# B&R Automation Studio project Robot_control
Automation Studio 4.8.2.72

## Configuration Config1

CPU X20CP1382, AutomationRuntime B4.82, Build 4.1.2, Vc V4.72.1

### Task classes (Cpu.sw)
```
Cyclic#1 (cycle 1000 us, tolerance 1000 us):
  Program <- Program.prg
  OpcUA <- OpcUA.prg
  TCPServer <- TCPServer.prg
Binaries: udbdef, FWRules, TCData, sysconf, Role, User, iomap, ashwd, asfw, arconfig, ashwac
Libraries: AsIecCon, AsOpcUac, AsOpcUas, AsTCP, AsBrStr, runtime, astime, standard
```

### Hardware
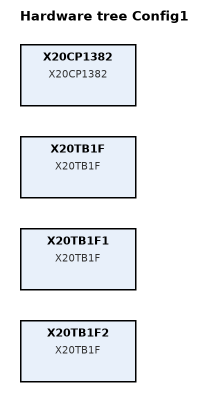
```
X20CP1382 : X20CP1382 v1.10.0.0  [X1 -> X1.SL; X2 -> X2.SL; X3 -> X3.SL]
  Module X1 (Type=X1, Virtual=true, Version=1.10.0.0)
    Connection (Connector=SS1, TargetModule=X20TB1F, TargetConnector=SS)
    Connection (Connector=SL, TargetModule=X20CP1382, TargetConnector=X1)
  Module X2 (Type=X2, Virtual=true, Version=1.10.0.0)
    Connection (Connector=SS1, TargetModule=X20TB1F1, TargetConnector=SS)
    Connection (Connector=SL, TargetModule=X20CP1382, TargetConnector=X2)
  Module X3 (Type=X3, Virtual=true, Version=1.10.0.0)
    Connection (Connector=SS1, TargetModule=X20TB1F2, TargetConnector=SS)
    Connection (Connector=SL, TargetModule=X20CP1382, TargetConnector=X3)
  Connector IF2:
    ActivateDevice = 1
    Mode = Manual
    InternetAddress = 192.168.0.20
    SubnetMask = 255.255.255.0
    ActivateSnmp = 2
  Connector IF7:
    Timeout = 1
  ConfigurationID = robot_control_Config1
  SystemTick = 1000
  TaskClassIdleTime = 1000
  Cyclic1Duration = 1000
  Cyclic1Tolerance = 1000
  Cyclic2Duration = 2000
  Cyclic2Tolerance = 2000
X20TB1F : X20TB1F v1.0.0.0
X20TB1F1 : X20TB1F v1.0.0.0
X20TB1F2 : X20TB1F v1.0.0.0
```

### IoMap.iom - X20CP1382/IoMap.iom
```iecst
VAR_CONFIG
	::Program:this.M1.direction AT %QX."X3".DigitalOutput04;
	::Program:this.M1.freq AT %QX."X3".DigitalOutput09;
	::Program:this.M2.direction AT %QX."X3".DigitalOutput05;
	::Program:this.M3.direction AT %QX."X3".DigitalOutput06;
	::Program:this.M2.freq AT %QX."X3".DigitalOutput10;
	::Program:this.M3.freq AT %QX."X3".DigitalOutput11;
	::Program:this.btn1.pressed AT %IX."X1".DigitalInput03;
	::Program:this.btn2.pressed AT %IX."X1".DigitalInput02;
	::Program:this.btn4.pressed AT %IX."X1".DigitalInput04;
	::Program:this.btn3.pressed AT %IX."X1".DigitalInput01;
	::Program:this.pencilSharp AT %QX."X3".DigitalOutput08;
	gNettime  AT %ID."X20CP1382".IF6.Nettime;
END_VAR
```

## Logical view

Binary libraries used (declarations not repeated): operator, runtime, astime, AsIecCon, AsOpcUac, AsOpcUas, AsTCP, AsBrStr, standard

### Global.typ
```iecst
TYPE
	coord_typ : 	STRUCT  (*Meant to be an array of coordinates*)
		z : DINT; (*Also called draw*)
		y : DINT;
		x : DINT;
	END_STRUCT;
END_TYPE
```

### Global.var
```iecst
VAR
	coord : ARRAY[0..LENGT_OF_COORD] OF coord_typ;
	gNettime : DINT;
	pSharp : BOOL;
	draw_old : DINT;
	draw : DINT := 0;
	y_coord : DINT := 0;
	x_coord : DINT := 0;
	goTo : STRING[80];
END_VAR
(*SPEED : TIME;*)
(*Global constants*)
VAR CONSTANT
	LENGT_OF_COORD : USINT := 200; (*maximum number of stored coords*)
END_VAR
```

### Program Logical/OpcUA

#### Types.typ
```iecst
TYPE
	OPC :
		(
		OPC_START_OPERATE,
		OPC_METHOD_CALLED,
		OPC_METHOD_EXECUTE,
		OPC_FINISH_OPERATE,
		OPC_FINISH_METHOD,
		OPC_ERROR
		);
END_TYPE
```

#### Variables.var
```iecst
VAR
	lookAt : USINT;
	result : USINT;
	ma : USINT;
	mb : USINT;
	UaSrv_MethodOperate_0 : UaSrv_MethodOperate;
	stOpcMethod : OPC;
	errorID : DWORD;
END_VAR
```

#### Main.st
```iecst
PROGRAM _INIT

END_PROGRAM

PROGRAM _CYCLIC
	CASE stOpcMethod OF
		OPC_START_OPERATE: // start operate
			UaSrv_MethodOperate_0.Action  := UaMoa_CheckIsCalled;
			UaSrv_MethodOperate_0.MethodName := 'Multiply';
			UaSrv_MethodOperate_0.Execute := TRUE;
			stOpcMethod := OPC_METHOD_CALLED;
		OPC_METHOD_CALLED: // check if method called
			UaSrv_MethodOperate_0();
			IF UaSrv_MethodOperate_0.Busy THEN
				UaSrv_MethodOperate_0.Execute := FALSE;
			ELSE
				IF UaSrv_MethodOperate_0.Done THEN
					errorID := 0;
					IF UaSrv_MethodOperate_0.IsCalled THEN
						stOpcMethod := OPC_METHOD_EXECUTE; // method is called
					END_IF
					UaSrv_MethodOperate_0.Execute := TRUE;
				END_IF
				IF UaSrv_MethodOperate_0.Error THEN
					errorID:= UaSrv_MethodOperate_0.ErrorID;
					stOpcMethod := OPC_ERROR;
				END_IF
			END_IF
		OPC_METHOD_EXECUTE: // execute method code
			result := ma * mb;
			stOpcMethod := OPC_FINISH_OPERATE;
		OPC_FINISH_OPERATE: // finish operate
			UaSrv_MethodOperate_0.Action  := UaMoa_Finished;
			UaSrv_MethodOperate_0.MethodName := 'Multiply';
			UaSrv_MethodOperate_0.Execute := TRUE;
			stOpcMethod := OPC_FINISH_METHOD;
		OPC_FINISH_METHOD: // finish method
			UaSrv_MethodOperate_0();
			IF UaSrv_MethodOperate_0.Busy THEN
				UaSrv_MethodOperate_0.Execute := FALSE;
			ELSE
				IF UaSrv_MethodOperate_0.Done THEN
					errorID:= 0;
					stOpcMethod := OPC_START_OPERATE; // method is finished, wait again for call
				END_IF
				IF UaSrv_MethodOperate_0.Error THEN
					errorID:= UaSrv_MethodOperate_0.ErrorID;
					stOpcMethod := OPC_ERROR;
				END_IF
			END_IF
	END_CASE;
END_PROGRAM

PROGRAM _EXIT

END_PROGRAM
```

- Methods.uam (not shown)

### Program Logical/Program (IEC)

#### Main.st - Init, cyclic, exit code
```iecst
PROGRAM _INIT
	draw := 5;
	this.start := TRUE;
	this.topSpeed 		:= T#0ms; 	// This parameter will slow the topspeed of all axis.
	this.acceleration	:= 1;		// This parameter will smoothen the acceleration of all axis.

END_PROGRAM

PROGRAM _CYCLIC
	(**********************************************************************************************)
	(************************************** Startup sequence **************************************)
	(**********************************************************************************************)
	IF this.start AND gNettime <> 0 THEN
		CASE this.startCase OF
			0: // First find M3 and M2 home switch
				this.M3.backward 	:= TRUE;
				this.M2.backward 	:= TRUE;

				IF this.btn3.pressed THEN
					this.M1.backward:= TRUE;
					this.startCase 	:= 10;
				END_IF;

			10: // Waiting for M1 and M2 to be homed
				IF this.btn1.pressed THEN
					this.M1.counter	:= 0;
				END_IF;

				IF this.btn2.pressed THEN
					this.M2.counter := 0;
				END_IF;

				IF this.btn1.pressed AND this.btn2.pressed THEN
					this.startCase := 15;
				END_IF;

			15:// going to origo (0,0)
				IF this.M1.counter < 4000 THEN
					this.M1.forward := TRUE;
				ELSE
					this.M1.forward := FALSE;
				END_IF;

				IF this.M2.counter < 275 THEN
					this.M2.forward := TRUE;
				ELSE
					this.M2.forward := FALSE;
				END_IF;

				IF this.M1.counter >= 4000 AND this.M2.counter >= 275 THEN
					this.startCase := 20;
				END_IF;

			20: // make sure the pencil have reached origo with M3
				IF this.btn4.pressed THEN
					this.startCase := 25;
				ELSE
					this.M3.forward := TRUE;
				END_IF;

			25: // Set all counter values to 0
				this.M1.counter := 0;
				this.M2.counter := 0;
				this.M3.counter := 0;
				this.startCase := 30;

			30: // Lift the pencil from the paper again
				IF this.M3.counter > -500 THEN
					this.M3.backward := TRUE;
				ELSE
					this.M3.backward := FALSE;
					this.startCase := 35;
				END_IF;

			35: // Ready to start drawing
				this.start 		:= FALSE;
				this.startCase 	:= FALSE;
				this.isReady 	:= TRUE;

		END_CASE;
	END_IF

	(**********************************************************************************************)
	(*********************************** Coordinate translation ***********************************)
	(**********************************************************************************************)
	// Read and translate the coordinates from java server
	IF NOT pSharp THEN
		CASE case_draw OF
			0: // start the case
				IF coord[LENGT_OF_COORD].x <> -1 AND coord[LENGT_OF_COORD].y <> -1 AND coord[LENGT_OF_COORD].z <> -1 THEN
					this.coord.x := coord[LENGT_OF_COORD].x;
					this.coord.y := coord[LENGT_OF_COORD].y;
					this.coord.z := coord[LENGT_OF_COORD].z;
					coord[LENGT_OF_COORD].x := -1;
					coord[LENGT_OF_COORD].y := -1;
					coord[LENGT_OF_COORD].z := -1;
					case_draw := 5;
				END_IF

			5: // which height should we goto?
				IF this.coord.z = 0 THEN // Black
					this.M3.goToCounter := 110;
					this.M3.goTo 		:= TRUE;
				ELSIF this.coord.z = 1 THEN
					this.M3.goToCounter := 75;
					this.M3.goTo 		:= TRUE;
				ELSIF this.coord.z = 2 THEN
					this.M3.goToCounter := 30;
					this.M3.goTo 		:= TRUE;
				ELSIF this.coord.z = 3 THEN
					this.M3.goToCounter := -65;
					this.M3.goTo 		:= TRUE;
				ELSIF this.coord.z = 4 THEN
					this.M3.goToCounter := -75;
					this.M3.goTo 		:= TRUE;
				ELSIF this.coord.z = 5 THEN // White
					this.M3.goToCounter := -200;
					this.M3.goTo 		:= TRUE;
				END_IF

				IF this.M3.counter = this.M3.goToCounter THEN
					case_draw := 10;
				END_IF

			10: // Goto all the coordinates, and then go back to state 0 to calculate next coordinate
				this.M1.goToCounter := this.coord.x * 40;
				this.M2.goToCounter := this.coord.y * 40;
				this.M1.goTo := TRUE;
				this.M2.goTo := TRUE;
				IF this.M3.counter <> this.M3.goToCounter THEN
					this.M3.goTo := TRUE;
				END_IF

				IF (this.M1.goToCounter = this.M1.counter AND this.M2.goToCounter = this.M2.counter AND this.M3.goToCounter = this.M3.counter) THEN
					case_draw := 0;
				END_IF

		END_CASE;
	END_IF;

	(**********************************************************************************************)
	(*********************************** Pencil sharpener logic ***********************************)
	(**********************************************************************************************)
	// Controls the acceleration when pencil sharpening
	IF EDGEPOS(pSharp) AND this.acceleration < 2 THEN
		this.acceleration 			:= this.acceleration + 2;
		this.accelerationChangePS 	:= TRUE;
	ELSIF EDGENEG(pSharp) AND this.accelerationChangePS THEN
		this.acceleration			:= this.acceleration - 2;
		this.accelerationChangePS	:= FALSE;
	END_IF

	// Calculate when to sharp the pencil
	// No wear on the pencil when draw value is 5
	// Approx. 175000 ms if the pencil draw value is 4
	// Approx. 164000 ms if the pencil draw value is 3
	// Approx. 150000 ms if the pencil draw value is 2
	// Approx. 130000 ms if the pencil draw value is 1
	// Approx. 100000 ms if the pencil draw value is 0
	IF this.coord.x > 0 AND this.coord.y > 0 AND this.coord.z > 0 THEN
		IF draw = 4 THEN
			dull_counter := dull_counter + 1;
		ELSIF draw = 3 THEN
			dull_counter := dull_counter + 1.06;
		ELSIF draw = 2 THEN
			dull_counter := dull_counter + 1.16;
		ELSIF draw = 1 THEN
			dull_counter := dull_counter + 1.35;
		ELSIF draw = 0 THEN
			dull_counter := dull_counter + 1.75;
		END_IF
	END_IF

	IF (dull_counter > 175000) THEN
		pSharp := TRUE;
		dull_counter := 0;
		this.startPS := TRUE;
	END_IF;

	IF this.startPS THEN // When the dull counter runs out, pencil sharpener case starts
		CASE this.startPSCase OF
			0: // Store goTo values
				this.M1.goToCounter := this.M1.counter;
				this.M3.goToCounter := this.M3.counter;
				this.m3TempPS		:= this.M3.counter;
				this.startPSCase := 5;

			5: // lift the pencil from the drawing plane, and go to an height that fits the pencil sharpener
				this.M3.backward := TRUE;

				IF this.M3.counter < -200 AND this.M1.counter > -2500 THEN
					this.M1.backward := TRUE;
				ELSE
					this.M1.backward := FALSE;
				END_IF

				IF this.M3.counter = -3200 THEN
					this.M3.backward := FALSE;
					this.startPSCase := 10;
				END_IF

			10: // Start moving towards the pencil sharpener, and wait for switch above pencil sharpener to be activated
				this.M1.backward := TRUE;
				IF this.btn1.pressed THEN
					this.M1.backward := FALSE;
					this.startPSCase := 15;
				END_IF

			15: // start pencil sharpener, and go into the pencil sharpener
				this.pencilSharp := TRUE;
				this.M3.goToCounter := 110;
				this.M3.goTo := TRUE;

				IF EDGEPOS(this.btn4.pressed)THEN
					this.M3.counter	:= 0;
				END_IF

				IF this.btn4.pressed THEN
					sharp_counter := sharp_counter +1;
				END_IF

				IF sharp_counter > 500 THEN // go deeper
					sharp_counter := 0;
					this.startPSCase := 16;
				END_IF;

			16: // start going deeper
				this.M3.goToCounter := 130;
				this.M3.goTo := TRUE;
				sharp_counter := sharp_counter +1;

				IF sharp_counter > 500 THEN // go deeper
					sharp_counter := 0;
					this.startPSCase := 17;
				END_IF;

			17: // start going deeper
				this.M3.goToCounter := 145;
				this.M3.goTo := TRUE;
				sharp_counter := sharp_counter +1;

				IF sharp_counter > 3000 THEN // retreat
					sharp_counter := 0;
					this.startPSCase := 20;
				END_IF;

			20: // move out of the pencil sharpener
				this.M3.backward := TRUE;

				IF this.M3.counter = -1950 THEN
					this.M3.backward := FALSE;
					this.startPSCase := 25;
					this.pencilSharp := FALSE;
				END_IF

			25: // move back to position
				this.M1.goTo := TRUE;

				IF this.M1.counter > - 2800 THEN
					this.M3.goToCounter := 800;
					this.M3.goTo 		:= TRUE;
					this.startPSCase 	:= 27;
				END_IF

			27: // Calibrate axis 3 on the drawining plane
				IF this.M1.goTo = FALSE AND this.M3.goTo = FALSE THEN
					this.M3.forward := TRUE;
				END_IF

				IF this.btn4.pressed THEN
					this.M3.counter 	:= 0;
					this.M3.forward		:= FALSE;
					this.startPSCase 	:= 30;
				END_IF

			30: // go to the correct heigt
				IF this.M1.goTo = FALSE THEN
					this.M3.goToCounter := this.m3TempPS;
					this.M3.goTo := TRUE;
					this.startPSCase := 35;
				END_IF

			35: // Continues from where it left
				this.startPS := FALSE;
				this.startPSCase := 0;
				pSharp := FALSE;

		END_CASE
	END_IF

	(**********************************************************************************************)
	(****************************************** Subcasses *****************************************)
	(**********************************************************************************************)
	M1_speedCase;
	M2_speedCase;
	M3_speedCase;

END_PROGRAM
```

#### Types.typ - Local data types
```iecst
TYPE
	m_typ : 	STRUCT  (*Types used for all motors*)
		endSwitch : BOOL;
		freq : BOOL; (*Output frequency for the steppermotor*)
		backward : BOOL; (*Backward movement towards the switch when true*)
		forward : BOOL; (*Forward movement when true*)
		direction : BOOL; (*Output direction for the steppermotor*)
		counter : DINT; (*Actual position*)
		goTo : BOOL; (*When true, the axis will goTo the goToCounter value*)
		goToCounter : DINT; (*The postion the axis should go to*)
		speedCaseTON : TON; (*Used to control acceleration*)
		speedCase : USINT; (*Used to control acceleration*)
		overRideCase : USINT; (*This case is used if you want to go further than the endswitch*)
	END_STRUCT;
	this_typ : 	STRUCT  (*Local structure type*)
		M1 : m_typ;
		M2 : m_typ;
		M3 : m_typ;
		topSpeed : TIME; (*T#0ms = 1 bit every 1 ms, T#5ms = 1 bit every 5 ms*)
		acceleration : USINT; (*0 = instant topspeed, 10 = slowest acceleration*)
		btn2 : btn_typ;
		isReady : BOOL;
		btn4 : btn_typ;
		btn3 : btn_typ;
		btn1 : btn_typ;
		startCase : USINT;
		start : BOOL;
		startPSCase : USINT;
		startPS : BOOL;
		accelerationChangePS : BOOL; (*If the acceleration have been changed when pencil sharpening, then this bool will be true*)
		m3TempPS : DINT;
		pencilSharp : BOOL;
		greyScale : USINT;
		print : BOOL; (*If print is equal to 1 then it should be printing*)
		coord : coord_typ;
	END_STRUCT;
	btn_typ : 	STRUCT
		pressed : BOOL;
	END_STRUCT;
END_TYPE
```

#### Variables.var - Local variables
```iecst
VAR
	dull_counter : REAL;
	sharp_counter : DINT;
	case_draw : USINT;
	this : this_typ;
END_VAR
```

#### M1_speedCase.st
```iecst
ACTION M1_speedCase:

	CASE this.M1.speedCase OF
		0: // highest speed
			this.M1.speedCaseTON.PT := this.topSpeed;

		1:
			this.M1.speedCaseTON.PT := this.topSpeed + T#1ms;

		2:
			this.M1.speedCaseTON.PT := this.topSpeed + T#2ms;

		3:
			this.M1.speedCaseTON.PT := this.topSpeed + T#3ms;

		4:
			this.M1.speedCaseTON.PT := this.topSpeed + T#4ms;

		5:
			this.M1.speedCaseTON.PT := this.topSpeed + T#5ms;

		6:
			this.M1.speedCaseTON.PT := this.topSpeed + T#6ms;

		7:
			this.M1.speedCaseTON.PT := this.topSpeed + T#7ms;

		8:
			this.M1.speedCaseTON.PT := this.topSpeed + T#8ms;

		9:
			this.M1.speedCaseTON.PT := this.topSpeed + T#9ms;

		10:
			this.M1.speedCaseTON.PT := this.topSpeed + T#10ms;

	END_CASE

	IF this.M1.forward OR this.M1.backward THEN
		IF this.M1.speedCaseTON.Q THEN
			this.M1.speedCaseTON.IN := FALSE;

			IF this.M1.freq THEN
				this.M1.freq 		:= FALSE;
			ELSE
				this.M1.freq		:= TRUE;
			END_IF

		ELSE
			this.M1.speedCaseTON.IN := TRUE;

		END_IF
	END_IF

	IF this.M1.forward THEN
		this.M1.direction := TRUE;

		IF EDGEPOS(this.M1.freq) THEN
			this.M1.counter := this.M1.counter + 1;

			IF this.M1.speedCase > 0 THEN
				this.M1.speedCase := this.M1.speedCase - 1;
			END_IF

		ELSIF EDGEPOS(NOT(this.M1.freq)) THEN
			this.M1.counter := this.M1.counter + 1;
		END_IF;
	ELSIF this.M1.backward THEN
		this.M1.direction := FALSE;

		IF EDGEPOS(this.M1.freq) THEN
			this.M1.counter := this.M1.counter - 1;

			IF this.M1.speedCase > 0 THEN
				this.M1.speedCase := this.M1.speedCase - 1;
			END_IF

		ELSIF EDGEPOS(NOT(this.M1.freq)) THEN
			this.M1.counter := this.M1.counter - 1;
		END_IF;

	END_IF
	IF EDGEPOS(NOT(this.M1.backward)) OR EDGEPOS(NOT(this.M1.forward)) THEN
		this.M1.speedCase := this.acceleration;

	END_IF

	this.M1.speedCaseTON ();
END_ACTION
```

#### M2_speedCase.st
```iecst
ACTION M2_speedCase:

	CASE this.M2.speedCase OF
		0: // highest speed
			this.M2.speedCaseTON.PT := this.topSpeed;

		1:
			this.M2.speedCaseTON.PT := this.topSpeed + T#1ms;

		2:
			this.M2.speedCaseTON.PT := this.topSpeed + T#2ms;

		3:
			this.M2.speedCaseTON.PT := this.topSpeed + T#3ms;

		4:
			this.M2.speedCaseTON.PT := this.topSpeed + T#4ms;

		5:
			this.M2.speedCaseTON.PT := this.topSpeed + T#5ms;

		6:
			this.M2.speedCaseTON.PT := this.topSpeed + T#6ms;

		7:
			this.M2.speedCaseTON.PT := this.topSpeed + T#7ms;

		8:
			this.M2.speedCaseTON.PT := this.topSpeed + T#8ms;

		9:
			this.M2.speedCaseTON.PT := this.topSpeed + T#9ms;

		10:
			this.M2.speedCaseTON.PT := this.topSpeed + T#10ms;

	END_CASE

	IF this.M2.forward OR this.M2.backward THEN
		IF this.M2.speedCaseTON.Q THEN
			this.M2.speedCaseTON.IN := FALSE;

			IF this.M2.freq THEN
				this.M2.freq 		:= FALSE;
			ELSE
				this.M2.freq		:= TRUE;
			END_IF

		ELSE
			this.M2.speedCaseTON.IN := TRUE;

		END_IF
	END_IF

	IF this.M2.forward THEN // Logic for acceleration
		this.M2.direction := TRUE;

		IF EDGEPOS(this.M2.freq) THEN
			this.M2.counter := this.M2.counter + 1;

			IF this.M2.speedCase > 0 THEN
				this.M2.speedCase := this.M2.speedCase - 1;
			END_IF

		ELSIF EDGEPOS(NOT(this.M2.freq)) THEN
			this.M2.counter := this.M2.counter + 1;
		END_IF;
	ELSIF this.M2.backward THEN
		this.M2.direction := FALSE;

		IF EDGEPOS(this.M2.freq) THEN
			this.M2.counter := this.M2.counter - 1;

			IF this.M2.speedCase > 0 THEN
				this.M2.speedCase := this.M2.speedCase - 1;
			END_IF

		ELSIF EDGEPOS(NOT(this.M2.freq)) THEN
			this.M2.counter := this.M2.counter - 1;
		END_IF;

	END_IF
	IF EDGEPOS(NOT(this.M2.backward)) OR EDGEPOS(NOT(this.M2.forward)) THEN
		this.M2.speedCase := this.acceleration;

	END_IF

	// Logic for goto
	IF this.M2.goTo AND (this.M2.goToCounter <> this.M2.counter) THEN
		IF this.M2.counter < this.M2.goToCounter THEN
			this.M2.forward := TRUE;
			this.M2.backward := FALSE;
		ELSIF this.M2.counter > this.M2.goToCounter THEN
			this.M2.backward := TRUE;
			this.M2.forward := FALSE;
		END_IF
	ELSIF this.M2.goTo AND (this.M2.goToCounter = this.M2.counter) THEN
		this.M2.backward := FALSE;
		this.M2.forward := FALSE;
		this.M2.goTo := FALSE;
	END_IF

	// Safety feature
	IF this.btn2.pressed THEN
		this.M2.backward := FALSE;
	END_IF;

	this.M2.speedCaseTON ();

END_ACTION
```

#### M3_speedCase.st
```iecst
ACTION M3_speedCase:

	CASE this.M3.speedCase OF
		0: // highest speed
			this.M3.speedCaseTON.PT := this.topSpeed;

		1:
			this.M3.speedCaseTON.PT := this.topSpeed + T#1ms;

		2:
			this.M3.speedCaseTON.PT := this.topSpeed + T#2ms;

		3:
			this.M3.speedCaseTON.PT := this.topSpeed + T#3ms;

		4:
			this.M3.speedCaseTON.PT := this.topSpeed + T#4ms;

		5:
			this.M3.speedCaseTON.PT := this.topSpeed + T#5ms;

		6:
			this.M3.speedCaseTON.PT := this.topSpeed + T#6ms;

		7:
			this.M3.speedCaseTON.PT := this.topSpeed + T#7ms;

		8:
			this.M3.speedCaseTON.PT := this.topSpeed + T#8ms;

		9:
			this.M3.speedCaseTON.PT := this.topSpeed + T#9ms;

		10:
			this.M3.speedCaseTON.PT := this.topSpeed + T#10ms;

	END_CASE

	IF this.M3.forward OR this.M3.backward THEN
		IF this.M3.speedCaseTON.Q THEN
			this.M3.speedCaseTON.IN := FALSE;

			IF this.M3.freq THEN
				this.M3.freq 		:= FALSE;
			ELSE
				this.M3.freq		:= TRUE;
			END_IF

		ELSE
			this.M3.speedCaseTON.IN := TRUE;

		END_IF
	END_IF

	IF this.M3.forward THEN
		this.M3.direction := TRUE;

		IF EDGEPOS(this.M3.freq) THEN
			this.M3.counter := this.M3.counter + 1;

			IF this.M3.speedCase > 0 THEN
				this.M3.speedCase := this.M3.speedCase - 1;
			END_IF

		ELSIF EDGEPOS(NOT(this.M3.freq)) THEN
			this.M3.counter := this.M3.counter + 1;
		END_IF;
	ELSIF this.M3.backward THEN
		this.M3.direction := FALSE;

		IF EDGEPOS(this.M3.freq) THEN
			this.M3.counter := this.M3.counter - 1;

			IF this.M3.speedCase > 0 THEN
				this.M3.speedCase := this.M3.speedCase - 1;
			END_IF

		ELSIF EDGEPOS(NOT(this.M3.freq)) THEN
			this.M3.counter := this.M3.counter - 1;
		END_IF;

	END_IF
	IF EDGEPOS(NOT(this.M3.backward)) OR EDGEPOS(NOT(this.M3.forward)) THEN
		this.M3.speedCase := this.acceleration;

	END_IF

	this.M3.speedCaseTON ();
END_ACTION
```

#### Action.st - not listed in the package file held
```iecst
ACTION LocalArrayAction:

	localArray1[0] := localArray.0;
	localArray1[1] := localArray.1;
	localArray1[2] := localArray.2;
	localArray1[3] := localArray.3;
	localArray1[4] := localArray.4;
	localArray1[5] := localArray.5;
	localArray1[6] := localArray.6;
	localArray1[7] := localArray.7;
	localArray1[8] := localArray.8;
	localArray1[9] := localArray.9;
	localArray1[10] := localArray.10;
	localArray1[11] := localArray.11;
	localArray1[12] := localArray.12;
	localArray1[13] := localArray.13;
	localArray1[14] := localArray.14;
	localArray1[15] := localArray.15;

END_ACTION
```

### Program Logical/TCPServer (IEC)

#### Main.st - Init, cyclic, exit code
```iecst
PROGRAM _INIT
	tcpst := TCPSTATE_SOCKET_OPEN;
	coord_counter := 1;

	FOR i:= 0 TO LENGT_OF_COORD DO 	// We do not have coordinates with values lower than 0,
		coord[i].x := -1;  			// that is why we set the init values to -1, to recognize
		coord[i].y := -1;			// the empty coordinates
		coord[i].z := -1;
	END_FOR;

END_PROGRAM

PROGRAM _CYCLIC
	IF (coord[1].x = -1 AND coord[1].y = -1 AND coord[1].z = -1) OR		// This if statement, makes sure that we will not fill the array
		(coord[3].x = -1 AND coord[3].y = -1 AND coord[3].z = -1) THEN 	// and keep getting new coordinates, with nowhere to store them.
	CASE tcpst OF
		TCPSTATE_SOCKET_OPEN :
			TcpOpen1.enable := TRUE;
			TcpOpen1.port := 2050;
			TcpOpen1.options := tcpOPT_REUSEADDR;
			TcpOpen1();
			IF (TcpOpen1.status = ERR_OK) THEN
				tcpst := TCPSTATE_SERVER_CREATE;
			END_IF

		TCPSTATE_SERVER_CREATE :
			IF goTo = sendData AND goTo = receiveData AND goTo <> '' THEN
				IF coord_counter = 1 THEN
					x_coord := brsatoi(ADR(goTo));
					goTo := '';
				ELSIF coord_counter = 2 THEN
					y_coord := brsatoi(ADR(goTo));
					goTo := '';
				ELSIF coord_counter = 3 THEN
					draw := brsatoi(ADR(goTo));
					goTo := '';
				END_IF
				sendData := receiveData := '';
				// goTo := '';
				coord_counter := coord_counter + 1;
				IF coord_counter >= 4 AND coord[0].x = -1 AND coord[0].y = -1 AND coord[0].z = -1 THEN
					coord[0].x := x_coord;
					coord[0].y := y_coord;
					coord[0].z := draw;
					coord_counter := 1;
					goTo := 'done';
				END_IF
			END_IF;

			TcpServer1.enable := TRUE;
			TcpServer1.ident := TcpOpen1.ident;
			TcpServer1();

			IF goTo = 'done' AND (TcpServer1.status = ERR_OK) THEN
				sendData := goTo;
				// goTo := '';
				tcpst := TCPSTATE_SEND;
			ELSIF (TcpServer1.status = ERR_OK) THEN
				tcpst := TCPSTATE_RECEIVE;
			END_IF

		TCPSTATE_RECEIVE :
			TcpReceive1.enable := TRUE;
			TcpReceive1.ident := TcpServer1.identclnt;
			TcpReceive1.pData := ADR(receiveData);
			TcpReceive1.datamax := SIZEOF(receiveData);
			TcpReceive1();
			IF (TcpReceive1.status = ERR_OK) THEN
				tcpst := TCPSTATE_SEND;
				sendData := receiveData;
			END_IF

		TCPSTATE_SEND :
			TcpSend1.enable := TRUE;
			TcpSend1.ident := TcpServer1.identclnt;
			TcpSend1.pData := ADR(sendData);
			TcpSend1.datalen := brsstrlen(ADR(sendData));     // We use brsstrlen() to get the length in UDINT datatype
			TcpSend1();
			IF (TcpSend1.status = ERR_OK) THEN
				tcpst := TCPSTATE_CLOSE;
			END_IF

		TCPSTATE_CLOSE :
			goTo := sendData;
			IF sendData = 'done' THEN
				sendData := '';
			END_IF;
			TcpClose1.enable := TRUE;
			TcpClose1.ident := TcpServer1.identclnt;
			TcpClose1();
			IF (TcpClose1.status = ERR_OK) THEN
				test := FALSE;
				TcpServer1.enable := FALSE;
				TcpServer1();
				tcpst := TCPSTATE_SERVER_CREATE;
			END_IF

		END_CASE
	END_IF

	// This is the logic for a 'First In First Out' (FIFO) system
	FOR i := 1 TO LENGT_OF_COORD DO
		IF (coord[i].x = -1 AND coord[i].y = -1 AND coord[i].z = -1) AND 					// IF number i coordinates is empty
			(coord[i - 1].x <> -1 AND coord[i - 1].y <> -1 AND coord[i -1].z <> -1) THEN	// AND the number i - 1 has coordinates
			coord[i].x 		:= coord[i - 1].x;												// THEN move the i - 1 coordinates to i coordinates location
			coord[i].y 		:= coord[i - 1].y;
			coord[i].z 		:= coord[i - 1].z;
			coord[i - 1].x	:= -1;
			coord[i - 1].y	:= -1;
			coord[i - 1].z	:= -1;
		END_IF
	END_FOR;

END_PROGRAM
```

#### Types.typ - Local data types
```iecst
TYPE
	TCPSTATE :
		(
		TCPSTATE_SOCKET_OPEN,
		TCPSTATE_SERVER_CREATE,
		TCPSTATE_RECEIVE,
		TCPSTATE_SEND,
		TCPSTATE_CLOSE
	);
END_TYPE
```

#### Variables.var - Local variables
```iecst
VAR
	test : BOOL;
	i : INT;
	coord_counter : USINT;
	TcpClose2 : TcpClose;
	TcpClose1 : TcpClose;
	TcpSend1 : TcpSend;
	TcpReceive1 : TcpRecv;
	TcpServer1 : TcpServer;
	TcpOpen1 : TcpOpen;
	receiveData : STRING[80];
	sendData : STRING[80];
	tcpst : TCPSTATE;
END_VAR
```
